{attribute 'GeneratedUsingTerminal: EL2521--0000'}
{attribute addProperty BoxType "EL2521--0000"}
{attribute addProperty Id "InputsAT %I*Inputs_A33354244OutputsAT %Q*Outputs_8F8B60FA4WcStateAT %I*WcState_9091E0EB2InfoDataAT %I*InfoData_32EB74EA10"}
{attribute addProperty CRC "1758432863"}
{attribute addProperty Size "20"}
TYPE EL2521_68CF8E5F EXTENDS EtcSlaveTerminalBase_947E5A46 :
STRUCT
	{attribute addProperty Name "Inputs"}
	Inputs : Inputs_A3335424;
	{attribute addProperty Name "Outputs"}
	Outputs : Outputs_8F8B60FA;
	{attribute addProperty Name "WcState"}
	WcState : WcState_9091E0EB;
	{attribute addProperty Name "InfoData"}
	InfoData : InfoData_32EB74EA;
END_STRUCT
END_TYPE

(* stored: Version 1.2.0.0, ProductVersion 3.1.4024.9
   DUT EL2521_68CF8E5F: Id {a59ba739-6927-447b-83c5-7dab037436eb} *)
